// TIA Portal V18 export
DATA_BLOCK "RotPosCalc_DB"   // DB11
// stored: AutoNumber false, InstanceOfName Rot_Pos_Calc, InstanceOfType FB
"Rot_Pos_Calc"
   // VAR_INPUT
   //    PulsesPerRev : Int;
   //    Counts : DInt;
   //    UL_OF : Bool;
   //    LL_OF : Bool;
   //    StoppedTime : Time;
   //    RolloverValue : LReal;
   // END_VAR
   // VAR_OUTPUT
   //    RotPosAbsDeg : Real;
   //    RotPosRelDeg : Real;
   //    RotTurns : Real;
   //    Stopped : Bool;
   //    DirFwd : Bool;
   //    DirRev : Bool;
   //    DegPerCount : Real;
   // END_VAR
   // VAR_IN_OUT
   //    ZeroPos : Bool;
   //    LDSlot0_1 : Byte;
   //    Slot0 : Real;
   //    Slot1 : Real;
   // END_VAR
   // VAR
   //    PosAbsDegLReal : LReal;
   //    Static_1 : Real;
   //    LastEncCount : DInt;
   //    Stopped_TON { S7_SetPoint := 'True'} : TON_TIME;
   // END_VAR
BEGIN
END_DATA_BLOCK
